FUNCTION_BLOCK Plant
  (* Standard: 61499-2 *)
  (* Version 0.1, 2015-00-13, Th?o, PC_THEO *)
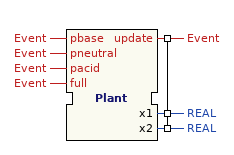
  EVENT_INPUT
    pbase;
    pneutral;
    pacid;
    full;
  END_EVENT
  EVENT_OUTPUT
    update WITH x1, x2;
  END_EVENT
  VAR_OUTPUT
    x1 : REAL;
    x2 : REAL;
  END_VAR
  VAR
    d : REAL;
  END_VAR
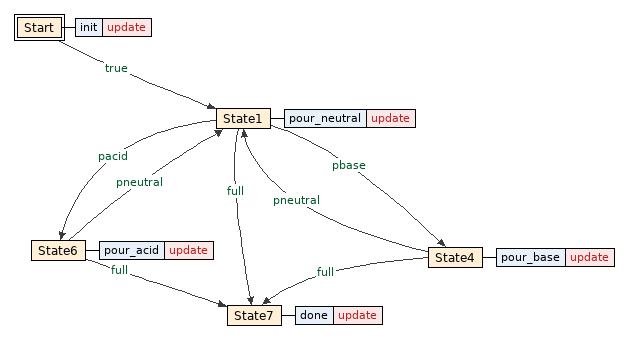
  EC_STATES
    Start : init -> update;
    State1 : pour_neutral -> update;
    State4 : pour_base -> update;
    State6 : pour_acid -> update;
    State7 : done -> update;
  END_STATES
  EC_TRANSITIONS
    Start TO State1 := true;
    State1 TO State7 := full;
    State1 TO State6 := pacid;
    State1 TO State4 := pbase;
    State4 TO State7 := full;
    State4 TO State1 := pneutral;
    State6 TO State7 := full;
    State6 TO State1 := pneutral;
  END_TRANSITIONS
  ALGORITHM init IN C:
me->x1=0.05;me->x2=7.1;
me->d=0.05;
printf("Initial pH : %f, Initial Volume : %f\n",me->x2, me->x1);
  END_ALGORITHM
  ALGORITHM pour_acid IN C:
//me->x1=me->x1+0.12*me->d;
//me->x2=me->x2-0.7*me->d;
me->x2=7.0;
me->x1=me->x1+me->d;
printf("Pouring acid, pH : %f, Volume : %f\n",me->x2, me->x1);
  END_ALGORITHM
  ALGORITHM pour_neutral IN C:
//me->x1=me->x1+0.1*me->d;
//me->x2=me->x2+0.1*me->d;
me->x2=7.205;
me->x1=me->x1+me->d;
printf("Pouring neutral, pH : %f, Volume : %f\n",me->x2, me->x1);
  END_ALGORITHM
  ALGORITHM pour_base IN C:
//me->x1=me->x1+0.12*me->d;
//me->x2=me->x2+0.9*me->d;
me->x2=7.0;
me->x1=me->x1+me->d;
printf("Pouring base, pH : %f, Volume : %f\n",me->x2, me->x1);
  END_ALGORITHM
  ALGORITHM done IN C:
printf("Tank full, pH : %f, Volume : %f\n",me->x2, me->x1);
  END_ALGORITHM
END_FUNCTION_BLOCK
